(* PLC project static_torsion.project, CODESYS CODESYS V3.5 SP17 Patch 3 *)
(* stored: creationDateTime 1970-01-01T00:00:00, modificationDateTime 2026-06-22T15:12:39.4699931 *)

TYPE S_STATE : STRUCT
  b0 : BIT;
  b1 : BIT;
  b2 : BIT;
  b3 : BIT;
  b4 : BIT;
  b5 : BIT;
  b6 : BIT;
  b7 : BIT;
  b8 : BIT;
  b9 : BIT;
  b10 : BIT;
  b11 : BIT;
  b12 : BIT;
  b13 : BIT;
  b14 : BIT;
  b15 : BIT;
END_STRUCT;
END_TYPE
